PROGRAM TEST_AXIS
VAR
  ncDelta : AXIS_REF;
  ncEcho : AXIS_REF;
	DELTA,ECHO: ROTAXIS_BECKHOFF;
	FOXTROTT: LINAXIS_JSC_XENAX;
END_VAR

FOXTROTT();
    DELTA(NCAxis := ncDelta);
    ECHO(NCAxis := ncEcho);

END_PROGRAM

(* stored: Version 1.1.0.1, ProductVersion 3.1.4026.18
   POU TEST_AXIS: Id {f1578d7a-8116-4732-8f15-c5150c9f53b8}, SpecialFunc None *)
